{attribute 'qualified_only'}
{attribute 'strict'}
{attribute 'to_string'}
TYPE ENUM_AxisStates :
(
    UNKNOWN := 0, // UNKNOWN must be in slot 0 or the FB breaks
    OUT := 1, 
    YAG := 2,
    TT := 3
) UINT;
END_TYPE

(* stored: Version 1.1.0.1
   DUT ENUM_AxisStates: Id {b411596a-bcb9-4bc6-9e2c-702c6c42053f} *)
